
// ===== library: MasterCopy "Özel Sayıcı" =====

FUNCTION_BLOCK "Özel Sayıcı"   // FB1, LAD
{ S7_Optimized_Access := 'TRUE' }
VERSION : 0.1
   VAR_INPUT
      ARTTIR : Bool;
      AZALT : Bool;
      ARTMA_MİKTARI : DInt;
      AZALMA_MİKTARI : DInt;
      ÜST_SINIR : DInt;
      ALT_SINIR : DInt;
      SİLME : Bool;
   END_VAR
   VAR_OUTPUT
      ÜST_ÇIKIŞ : Bool;
      ALT_ÇIKIŞ : Bool;
   END_VAR
   VAR_IN_OUT
      SAYICI_İÇERİĞİ : DInt;
   END_VAR
   VAR
      "ARTIŞ DARBE" : Bool;
      "AZALIŞ DARBE" : Bool;
   END_VAR
   VAR_TEMP   // added for the SCL form of the ladder/FBD networks
      _w1 : Bool;
   END_VAR
BEGIN

REGION Network 1
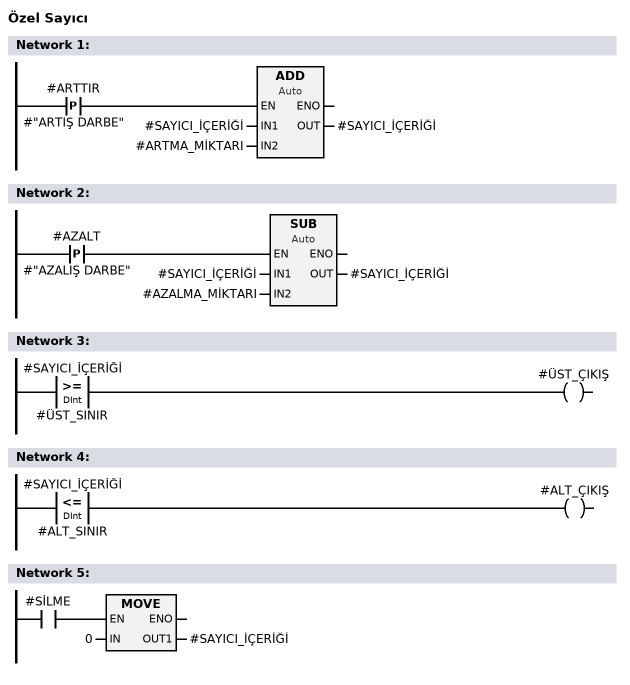
   RUNG wire#powerrail
      P_Contact(operand := #ARTTIR, bit := #"ARTIŞ DARBE")
      Add(in1 := #SAYICI_İÇERİĞİ, in2 := #ARTMA_MİKTARI, out => #SAYICI_İÇERİĞİ)
   END_RUNG
   // the same network as SCL:
   #_w1 := #ARTTIR AND NOT #"ARTIŞ DARBE";   // rising edge of #ARTTIR
   #"ARTIŞ DARBE" := #ARTTIR;
   IF #_w1 THEN #SAYICI_İÇERİĞİ := #SAYICI_İÇERİĞİ + #ARTMA_MİKTARI; END_IF;
END_REGION

REGION Network 2
   RUNG wire#powerrail
      P_Contact(operand := #AZALT, bit := #"AZALIŞ DARBE")
      Sub(in1 := #SAYICI_İÇERİĞİ, in2 := #AZALMA_MİKTARI, out => #SAYICI_İÇERİĞİ)
   END_RUNG
   // the same network as SCL:
   #_w1 := #AZALT AND NOT #"AZALIŞ DARBE";   // rising edge of #AZALT
   #"AZALIŞ DARBE" := #AZALT;
   IF #_w1 THEN #SAYICI_İÇERİĞİ := #SAYICI_İÇERİĞİ - #AZALMA_MİKTARI; END_IF;
END_REGION

REGION Network 3
   RUNG wire#powerrail
      { S7_Templates := "SrcType := DInt" } GE_Contact(in1 := #SAYICI_İÇERİĞİ, in2 := #ÜST_SINIR)
      Coil( #ÜST_ÇIKIŞ )
   END_RUNG
   // the same network as SCL:
   #ÜST_ÇIKIŞ := #SAYICI_İÇERİĞİ >= #ÜST_SINIR;
END_REGION

REGION Network 4
   RUNG wire#powerrail
      { S7_Templates := "SrcType := DInt" } LE_Contact(in1 := #SAYICI_İÇERİĞİ, in2 := #ALT_SINIR)
      Coil( #ALT_ÇIKIŞ )
   END_RUNG
   // the same network as SCL:
   #ALT_ÇIKIŞ := #SAYICI_İÇERİĞİ <= #ALT_SINIR;
END_REGION

REGION Network 5
   RUNG wire#powerrail
      Contact( #SİLME )
      Move(in := 0, out1 => #SAYICI_İÇERİĞİ)
   END_RUNG
   // the same network as SCL:
   IF #SİLME THEN #SAYICI_İÇERİĞİ := 0; END_IF;
END_REGION
END_FUNCTION_BLOCK